TEXTLIST St1AlarmList
  1 = 'a'
  2 = 'b'
   = ''
END_TEXTLIST

(* stored: Version 1.1.0.1
   TextList St1AlarmList: Id {e1f789a8-6b5c-490d-82e2-fb8d5dc61e93} *)
